{attribute 'reflection'}
FUNCTION_BLOCK PUBLIC FB_DevBase
VAR_INPUT
	nModuleId		: UDINT		:= 	1 					; // Higher level module ID
	bEnable			: BOOL 		:= TRUE 				; // Module enable signal reference Default := TRUE (when using system library := GVL_Main.stModules[nModuleId].bEnabled)
	bSafetyOk		: BOOL 		:= TRUE 				; // Module can operate safely [default true]
	bReset 			: BOOL 		:= FALSE				; // reset command bit reference Default := TRUE (when using system library := GVL_Main.stModules[nModuleId].bResetting)
	refFbFault		: REFERENCE TO Fb_FaultHandler	 	; // reference to fault handler ( when using utilities library := GVL_Main.stModules[nModuleId].fbFaultHandler)
	// function references 
	refFbManualCtrl	: REFERENCE TO FB_ManualController := GVL_DevManual.fbManualControler	; // reference to manual handler
	refFbParHandler	: REFERENCE TO Fb_ParLogging 	:= GVL_Parameters.fbParameterHandler	; // reference to parameter handler
END_VAR
VAR_IN_OUT
END_VAR
VAR_OUTPUT
	sDevActiveState	: STRING 		:= 'Idle'	; // active state of device 
	bInitOk			: BOOL 			:= FALSE 	; // function is initialized
	bBussy 			: BOOL 			:= FALSE 	; // device is busy
	bReady			: BOOL 			:= FALSE 	; // device is ready for new command 
	bManual			: BOOL 			:= false 	; // device is in manual mode
	bDevIsSafe		: BOOL 			:= FALSE	; // Device is locked and safe
	bErrorActive	: BOOL			:= FALSE	; // device Error active 
	bBlockedCommand	: BOOL 			:= False 	; // a device command is blocked because of collision detect 
	sDevName		: STRING 		; // Name of device distilled from the path 
	eDevType		: E_Devices	:= E_Devices.Undefined	; // Type of Device 	
	nDevNumber		: UDINT 		:= 0 		; // device sub number
	nDevId			: UDINT 		:= 0		; // device id number made up of module and device number				
END_VAR
VAR
	// Feedback request
	bMessageTest	: BOOL  		:= FALSE	; // Send test message from device
	// ===== Fault data =====
	stFault			: UDT_Fault	; // Fault data from device
	// Manual control variables
	bAddedToManual	: BOOL 			:= FALSE 	; // device is added tot manual control function 	
	bCmdManual 		: BOOL			:= FALSE	; // manual commands enabled control functions (thus disable automatic)
	// Function path 
	{attribute 'instance-path'} 
    {attribute 'noinit'}
	sPath			: STRING	; // Path name of function (used for manual reference)
END_VAR

ExecIdentifyDevice();

// Communicate active state
IF NOT bSafetyOk THEN 
	sDevActiveState := 'Safety not ok';
ELSIF bErrorActive THEN 
	sDevActiveState := TO_STRING(stFault.Discription);
ELSIF NOT bInitOk THEN 
	sDevActiveState := 'Not initialized';
ELSIF bManual THEN 
	sDevActiveState := 'Operational';
END_IF 

// Set fault if commands are blocked
IF bBlockedCommand THEN 
	stFault.Active 			:= TRUE ;
	stFault.ComponentType 	:= E_ComponentTypes.Assembly ;
	stFault.Discription		:= CONCAT( STR1 := sDevName, STR2 := 'Movement path is blocked');
	stFault.FaultType		:= E_FaultTypes.MC;
	refFbFault.CmdAddFault( stFault);
END_IF	
// Call reset function 
IF bReset THEN 
	CmdReset();
END_IF

METHOD PROTECTED CalcDeviceId : BOOL
VAR_INPUT
END_VAR
nDevId := (nModuleId * 10000) + nDevNumber * 100 ;
END_METHOD

METHOD PUBLIC CmdManual : BOOL
VAR_INPUT
END_VAR
bCmdManual := true ;
END_METHOD

METHOD CmdReset : BOOL
VAR_INPUT
END_VAR
END_METHOD

METHOD PUBLIC CmdSafeStop : BOOL
VAR_INPUT
END_VAR
// check if device is safe
bDevIsSafe 	:= NOT bEnable ;
CmdSafeStop := bDevIsSafe ;
END_METHOD

METHOD PRIVATE ExecIdentifyDevice : BOOL
VAR_INPUT
END_VAR
// Check device ID
IF bInitOk AND nDevId = 0 THEN 
	CalcDeviceId();
END_IF

// set message location information
stFault.LocationName	:= sDevName	;	
stFault.LocationNumber	:= nDevId	;

// Get device name from function and add device to manual
IF sDevName = '' THEN 
	sDevName := F_FBNameFromPath(sPath := sPath);
ELSIF NOT bAddedToManual AND eDevType <> E_Devices.Undefined THEN 
	bAddedToManual S= refFbManualCtrl.CmdAddDevice(THIS^);
END_IF

// Call message test function
ExecMessagTest();

bManual := bCmdManual ;
END_METHOD

METHOD ExecMessagTest : BOOL
VAR_INPUT
END_VAR
IF bMessageTest THEN 
	stFault.Active 			:= TRUE ;
	stFault.Discription 	:= CONCAT(STR1 := 'This is a test message from: ',STR2 := sDevName);
	stFault.MessageNumber 	:= E_MessageNumbers.OM_MessageTest ;
	stFault.FaultType		:= Utilities_Library.E_FaultTypes.OM ;
	refFbFault.CmdAddFault( stFault );
END_IF
END_METHOD

END_FUNCTION_BLOCK

(* stored: Version 1.1.0.1, ProductVersion 3.1.4024.4
   POU FB_DevBase: Id {fd1f0090-6070-4291-b370-d3eae943f30f}, SpecialFunc None
   Folder Private: Id {6f3beefb-a2d1-0bb4-3a9f-cd48592c8e20}
   Method CalcDeviceId: Id {821f405e-a996-09cf-2d6d-564182cfd77b}
   Method CmdManual: Id {26ba3ac1-09ba-01dd-32ca-9bbda4886bcd}
   Method CmdReset: Id {b56aa7b6-c59f-0fc2-1868-fb09dbbb1c2c}
   Method CmdSafeStop: Id {dec1b3af-006d-0b48-0f79-6a1440a93d4c}
   Method ExecIdentifyDevice: Id {54484a28-b20c-0028-16df-4783a8a55344}
   Method ExecMessagTest: Id {96681161-373a-0a03-14f8-0586e5796f7f} *)
